// TIA Portal V20 export
VAR_GLOBAL   // PLC tag table "BarcodeReader_DP3"
   "DP3-TriggerEnable" AT %Q223.0 : Bool;
   "DP3-Trigger" AT %Q223.1 : Bool;
   "DP3-TriggerReady" AT %I241.0 : Bool;
   "DP3-TriggerAck" AT %I241.1 : Bool;
   "DP3-Acquiring" AT %I241.2 : Bool;
   "DP3-MissedAcq" AT %I241.3 : Bool;
   "DP3-TriggerID" AT %IW242 : Word;
   "DP3-BufferResultsEnable" AT %Q224.0 : Bool;
   "DP3-ResultsAck" AT %Q224.1 : Bool;
   "DP3-Decoding" AT %I244.0 : Bool;
   "DP3-Decode Complete" AT %I244.1 : Bool;
   "DP3-Results Buffer Overrun" AT %I244.2 : Bool;
   "DP3-Results Available" AT %I244.3 : Bool;
   "DP3-General Fault" AT %I244.7 : Bool;
   "DP3-Train Code" AT %Q225.0 : Bool;
   "DP3-Train Match String" AT %Q225.1 : Bool;
   "DP3-Train Focus" AT %Q225.2 : Bool;
   "DP3-Train Brightness" AT %Q225.3 : Bool;
   "DP3-Untrain" AT %Q225.4 : Bool;
   "DP3-Execute DMCC" AT %Q225.6 : Bool;
   "DP3-Set Match String" AT %Q225.7 : Bool;
   "DP3-Train Code Ack" AT %I245.0 : Bool;
   "DP3-Train Match String Ack" AT %I245.1 : Bool;
   "DP3-Train Focus Ack" AT %I245.2 : Bool;
   "DP3-Train Brightness Ack" AT %I245.3 : Bool;
   "DP3-Untrain Ack" AT %I245.4 : Bool;
   "DP3-Execute DMCC Ack" AT %I245.6 : Bool;
   "DP3-Set Match String Ack" AT %I245.7 : Bool;
   "DP3-UserData Option" AT %QW226 : Word;
   "DP3-UserData Length" AT %QW228 : Word;
   "DP3-UserData[0]" AT %QB230 : Byte;
   "DP3-UserData[1]" AT %QB231 : Byte;
   "DP3-UserData[2]" AT %QB232 : Byte;
   "DP3-UserData[3]" AT %QB233 : Byte;
   "DP3-UserData[4]" AT %QB234 : Byte;
   "DP3-UserData[5]" AT %QB235 : Byte;
   "DP3-UserData[6]" AT %QB236 : Byte;
   "DP3-UserData[7]" AT %QB237 : Byte;
   "DP3-UserData[8]" AT %QB238 : Byte;
   "DP3-UserData[9]" AT %QB239 : Byte;
   "DP3-UserData[10]" AT %QB240 : Byte;
   "DP3-UserData[11]" AT %QB241 : Byte;
   "DP3-UserData[12]" AT %QB242 : Byte;
   "DP3-UserData[13]" AT %QB243 : Byte;
   "DP3-UserData[14]" AT %QB244 : Byte;
   "DP3-UserData[15]" AT %QB245 : Byte;
   "DP3-ResultID" AT %IW246 : Word;
   "DP3-Result Code" AT %IW249 : Word;
   "DP3-Read / No Read" AT %I249.0 : Bool;
   "DP3-Validated / Not Validated" AT %I249.1 : Bool;
   "DP3-Verified / Not Verified" AT %I249.2 : Bool;
   "DP3-Acquisition Trigger Overrun" AT %I249.3 : Bool;
   "DP3-Acquisition Buffer Overflow" AT %I249.4 : Bool;
   "DP3-Result Extended" AT %IW250 : Word;
   "DP3-Result Length" AT %IW252 : Word;
   "DP3-InspectionResults[0]" AT %IB254 : Byte;
   "DP3-InspectionResults[1]" AT %IB255 : Byte;
   "DP3-InspectionResults[2]" AT %IB256 : Byte;
   "DP3-InspectionResults[3]" AT %IB257 : Byte;
   "DP3-InspectionResults[4]" AT %IB258 : Byte;
   "DP3-InspectionResults[5]" AT %IB259 : Byte;
   "DP3-InspectionResults[6]" AT %IB260 : Byte;
   "DP3-InspectionResults[7]" AT %IB261 : Byte;
   "DP3-InspectionResults[8]" AT %IB262 : Byte;
   "DP3-InspectionResults[9]" AT %IB263 : Byte;
   "DP3-InspectionResults[10]" AT %IB264 : Byte;
   "DP3-InspectionResults[11]" AT %IB265 : Byte;
   "DP3-InspectionResults[12]" AT %IB266 : Byte;
   "DP3-InspectionResults[13]" AT %IB267 : Byte;
   "DP3-InspectionResults[14]" AT %IB268 : Byte;
   "DP3-InspectionResults[15]" AT %IB269 : Byte;
   "Result data_DP3" AT %I254.0 : "Global.BarCode";
   UserData_DP3 AT %Q230.0 : "Global.BarCode";
   ContinousGetResults_DP3 AT %M310.1 : Bool;
   TrainFocus_DP3 AT %M310.2 : Bool;
END_VAR
